Universal Robots PolyScope program: Test Square Motion.urp

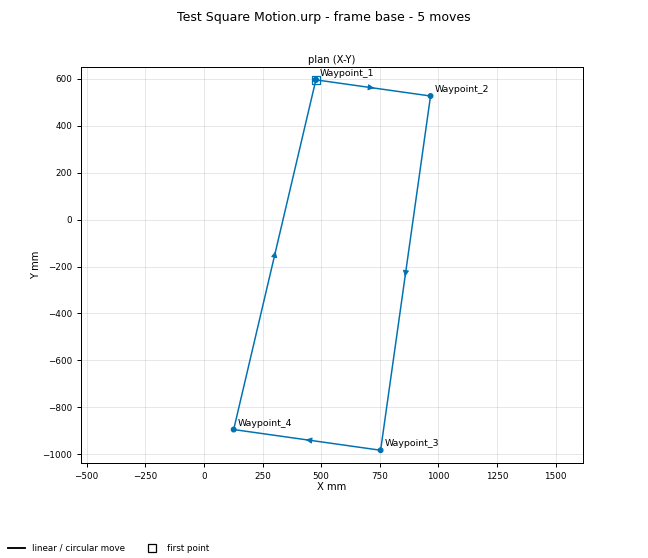
[picture p0: tool path of Test Square Motion.urp in frame base, 5 of 5 moves have a stored position in this frame; points joined in program order, loops and branches not executed]
Program Test Square Motion (installation=default directory=/programs createdIn=5.14.5 lastSavedIn=5.14.5 robotSerialNumber=20236801216)
Calibrated DH parameters: a=[-0.000021, -0.748897, -0.28186, -0.00004, -0.000055, 0]; d=[0.236225, -424.082933, -1564.66872, 1988.95162, 0.159094, 0.153873]; alpha=[1.570844, 0.001002, 0.000337, 1.571488, -1.569996, 0]; deltaTheta=[0, -0.516316, 5.626292, 1.173211, 0.000001, 0]
InitVariablesNode
Robot Program (runOnlyOnce=false)
  MoveL speed 250 mm/s, acceleration 1200 mm/s^2 (useActiveTCP=true) feature=Base
    Waypoint Waypoint_1: TCP in base x=477.467 y=596.236 z=273.467 mm, rx=-1.9895 ry=2.3598 rz=0.0268 rad; joints [66.618, -105.832, -136.829, -24.121, 89.513, 76.352] deg; TCP offset x=-0.005 y=-0.004 z=-0.034 mm, rx=0 ry=0 rz=0 rad
    Waypoint Waypoint_2: TCP in base x=966.474 y=527.332 z=273.447 mm, rx=-1.9895 ry=2.3598 rz=0.0268 rad; joints [38.946, -121.115, -108.576, -37.225, 91.097, 48.738] deg
    Waypoint Waypoint_3: TCP in base x=753.568 y=-983.519 z=273.45 mm, rx=-1.9895 ry=2.3598 rz=0.0268 rad; joints [-43.652, -127.736, -94.405, -48.55, 93.282, -33.904] deg
    Waypoint Waypoint_4: TCP in base x=126.89 y=-895.204 z=273.464 mm, rx=-1.9895 ry=2.3598 rz=0.0267 rad; joints [-69.594, -111.905, -123.963, -36.176, 92.66, -59.89] deg
    Waypoint Waypoint_1: TCP in base x=477.467 y=596.236 z=273.467 mm, rx=-1.9895 ry=2.3598 rz=0.0268 rad; joints [66.618, -105.832, -136.829, -24.121, 89.513, 76.352] deg
